{attribute 'qualified_only'}
{attribute 'strict'}
(*
Central definition of safety functions includes for a motion control cabinet.
Add new safety functions to match the incoming safety functions from the PNOZmulti 2.
Each safety function represents 4-bits of information. However the PLC still stores the incoming 4-bits
into 1-byte.
*)
TYPE E_SafetyFunctions:
(
    eNone,
    eEStop,
    eSampleStop,
    eSampleEnable,
    eDetectorArmIsolate,
    eDetectorEnable
);
END_TYPE

(* stored: Version 1.1.0.1
   DUT E_SafetyFunctions: Id {67cba4a1-d914-0ba8-3f98-b5150a554ddf} *)
